INTERFACE ITF_OpenDichtKlep

METHOD close : BOOL
VAR_INPUT
END_VAR
END_METHOD

METHOD open : BOOL
VAR_INPUT
END_VAR
END_METHOD

PROPERTY state : E_OpenDichtKlepState
GET
END_GET
END_PROPERTY

END_INTERFACE

(* stored: Version 1.1.0.1, ProductVersion 3.1.4024.13
   Itf ITF_OpenDichtKlep: Id {21e61fea-97d1-4c9c-b4fc-9ddab8b7f9d0}
   Method close: Id {f2f22f45-a88e-45a6-9f4a-e572e8906edd}
   Method open: Id {e548097a-12d8-4ea6-afe4-51826df3913b}
   Property state: Id {933d7d4e-6668-4e20-96e0-5e35819ba980}
   Get Get: Id {0bb3ceb1-3177-4442-abb1-eb5439853452} *)
